Universal Robots PolyScope program: test1.urp

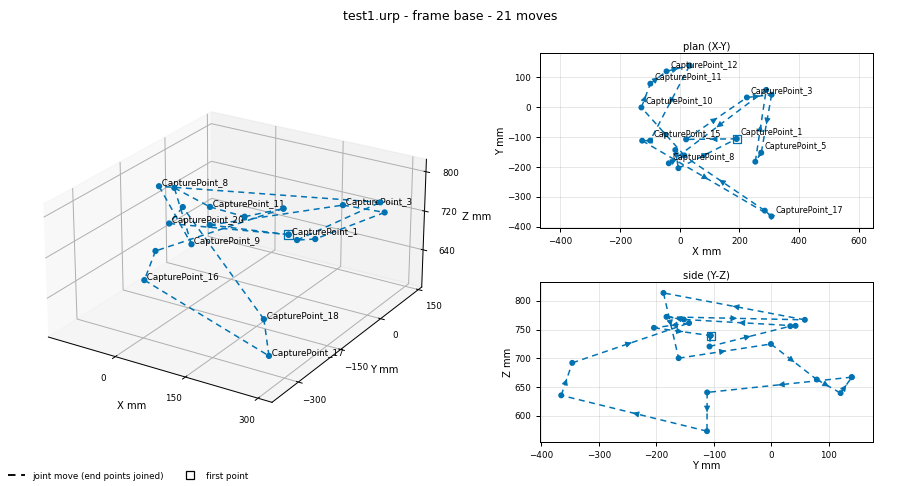
[picture p0: tool path of test1.urp in frame base, 21 of 21 moves have a stored position in this frame; points joined in program order, loops and branches not executed]
Program test1 (installation=default directory=/programs createdIn=3.8.0.61336 lastSavedIn=3.8.0.61336 robotSerialNumber=2018359174)
Calibrated DH parameters: a=[0.000103, -0.165236, -0.391809, -0.000008, 0.000072, 0]; d=[0.08937, 126.180413, -125.613724, -0.456703, 0.094787, 0.082637]; alpha=[1.569508, -0.003108, -0.027037, 1.57048, -1.570735, 0]; deltaTheta=[0, -1.172139, 1.133037, 0.038915, 0.000034, 0.000049]
Robot Program (runOnlyOnce=false)
  Script file /programs/X0.script
    | address="192.168.221.2"
    | port=3000
    | sname="mt"
    | socket_open(address,port,sname)
    | p=get_actual_tcp_pose()
    | socket_send_line("X0()",sname)
    | ret=socket_read_line(sname)
    | socket_close(sname)
    | if (ret != "OK"):
    |   popup(ret,title="X0",blocking=True)
    | end
  MoveJ speed 60 deg/s, acceleration 80 deg/s^2 (useActiveTCP=true)
    Waypoint CapturePoint_1: TCP in base x=190.534 y=-105.515 z=739.553 mm, rx=-2.169 ry=2.1248 rz=-0.0971 rad; joints [0.073, -70.662, -54.31, -138.22, 90.522, 0.198] deg
  Wait Sleep waitTime=1
  Script file /programs/X1.script
    | address="192.168.221.2"
    | port=3000
    | sname="mt"
    | socket_open(address,port,sname)
    | p=get_actual_tcp_pose()
    | rpy=rotvec2rpy([p[3],p[4],p[5]])
    | socket_send_string("X1(",sname)
    | socket_send_string(p[0]*1000.,sname)
    | socket_send_string(",",sname)
    | socket_send_string(p[1]*1000.,sname)
    | socket_send_string(",",sname)
    | socket_send_string(p[2]*1000.,sname)
    | socket_send_string(",",sname)
    | socket_send_string(r2d(rpy[0]),sname)
    | socket_send_string(",",sname)
    | socket_send_string(r2d(rpy[1]),sname)
    | socket_send_string(",",sname)
    | socket_send_string(r2d(rpy[2]),sname)
    | socket_send_line(")",sname)
    | ret=socket_read_line(sname)
    | socket_close(sname)
    | if (ret != "OK"):
    |   popup(ret,title="X1",blocking=True)
    | end
  MoveJ speed 60 deg/s, acceleration 80 deg/s^2 (useActiveTCP=true)
    Waypoint CapturePoint_2: TCP in base x=21.408 y=-107.346 z=720.582 mm, rx=-1.9877 ry=1.9105 rz=-0.2399 rad; joints [-30.105, -54.792, -66.384, -133.273, 107.073, -28.72] deg
  Wait Sleep waitTime=1
  Script file /programs/X1.script
    | (same text as the earlier copy of this file)
  MoveJ speed 60 deg/s, acceleration 80 deg/s^2 (useActiveTCP=true)
    Waypoint CapturePoint_3: TCP in base x=224.997 y=33.123 z=755.907 mm, rx=2.0802 ry=-2.0387 rz=0.3263 rad; joints [42.288, -80.135, -37.545, -164.25, 76.141, 44.096] deg
  Wait Sleep waitTime=1
  Script file /programs/X1.script
    | (same text as the earlier copy of this file)
  Wait Sleep waitTime=1
  MoveJ speed 60 deg/s, acceleration 80 deg/s^2 (useActiveTCP=true)
    Waypoint CapturePoint_4: TCP in base x=307.887 y=42.318 z=756.523 mm, rx=2.0137 ry=-1.9575 rz=0.3394 rad; joints [33.037, -92.913, -25.365, -167.152, 72.403, 35.309] deg
  Wait Sleep waitTime=1
  Script file /programs/X1.script
    | (same text as the earlier copy of this file)
  MoveJ speed 60 deg/s, acceleration 80 deg/s^2 (useActiveTCP=true)
    Waypoint CapturePoint_5: TCP in base x=273.105 y=-152.051 z=767.525 mm, rx=1.1431 ry=-2.8987 rz=-0.2387 rad; joints [-10.771, -92.914, -25.368, -157.055, 96.143, 37.312] deg
  Wait Sleep waitTime=1
  Script file /programs/X1.script
    | (same text as the earlier copy of this file)
  MoveJ speed 60 deg/s, acceleration 80 deg/s^2 (useActiveTCP=true)
    Waypoint CapturePoint_6: TCP in base x=253.251 y=-182.138 z=772.16 mm, rx=0.0328 ry=3.0997 rz=0.4007 rad; joints [-19.345, -92.915, -25.365, -155.309, 103.445, 72.846] deg
  Wait Sleep waitTime=1
  Script file /programs/X1.script
    | (same text as the earlier copy of this file)
  MoveJ speed 60 deg/s, acceleration 80 deg/s^2 (useActiveTCP=true)
    Waypoint CapturePoint_7: TCP in base x=289.745 y=58.466 z=766.928 mm, rx=2.7466 ry=0.3071 rz=0.0009 rad; joints [38.358, -91.191, -25.365, -165.797, 71.218, -60.862] deg
  Wait Sleep waitTime=1
  Script file /programs/X1.script
    | (same text as the earlier copy of this file)
  MoveJ speed 60 deg/s, acceleration 80 deg/s^2 (useActiveTCP=true)
    Waypoint CapturePoint_8: TCP in base x=-36.698 y=-187.426 z=813.704 mm, rx=-2.5132 ry=1.1035 rz=-0.5771 rad; joints [38.35, -58.013, -25.364, -158.36, 78.074, -5.557] deg
  Wait Sleep waitTime=1
  Script file /programs/X1.script
    | (same text as the earlier copy of this file)
  MoveJ speed 60 deg/s, acceleration 80 deg/s^2 (useActiveTCP=true)
    Waypoint CapturePoint_9: TCP in base x=15.55 y=-161.041 z=700.233 mm, rx=-2.5485 ry=1.1129 rz=-0.5577 rad; joints [43.689, -38.869, -67.087, -138.937, 75.373, -0.883] deg
  Wait Sleep waitTime=1
  Script file /programs/X1.script
    | (same text as the earlier copy of this file)
  MoveJ speed 60 deg/s, acceleration 80 deg/s^2 (useActiveTCP=true)
    Waypoint CapturePoint_10: TCP in base x=-128.422 y=-0.5 z=724.899 mm, rx=-1.2256 ry=2.2428 rz=-0.6001 rad; joints [-40.35, -38.871, -67.086, -127.735, 106.09, -0.879] deg
  Wait Sleep waitTime=1
  Script file /programs/X1.script
    | (same text as the earlier copy of this file)
  MoveJ speed 60 deg/s, acceleration 80 deg/s^2 (useActiveTCP=true)
    Waypoint CapturePoint_11: TCP in base x=-98.355 y=79.257 z=663.134 mm, rx=-0.6678 ry=2.3711 rz=-0.6414 rad; joints [-70.315, -30.072, -80.78, -124.448, 119.381, -0.99] deg
  Wait Sleep waitTime=1
  Script file /programs/X1.script
    | (same text as the earlier copy of this file)
  MoveJ speed 60 deg/s, acceleration 80 deg/s^2 (useActiveTCP=true)
    Waypoint CapturePoint_12: TCP in base x=-44.236 y=120.624 z=639.494 mm, rx=-0.028 ry=2.5208 rz=-0.5293 rad; joints [-97.846, -30.075, -80.778, -137.575, 123.899, -0.99] deg
  Wait Sleep waitTime=1
  Script file /programs/X1.script
    | (same text as the earlier copy of this file)
  MoveJ speed 60 deg/s, acceleration 80 deg/s^2 (useActiveTCP=true)
    Waypoint CapturePoint_13: TCP in base x=32.967 y=140.081 z=667.219 mm, rx=0.7689 ry=2.4403 rz=-0.2805 rad; joints [-127.955, -38.753, -66.496, -163.611, 124.333, -1.004] deg
  Wait Sleep waitTime=1
  Script file /programs/X1.script
    | (same text as the earlier copy of this file)
  MoveJ speed 60 deg/s, acceleration 80 deg/s^2 (useActiveTCP=true)
    Waypoint CapturePoint_14: TCP in base x=32.955 y=140.061 z=667.229 mm, rx=-1.0077 ry=2.5472 rz=-0.74 rad; joints [-127.955, -38.755, -66.496, -163.608, 124.335, -79.153] deg
  Wait Sleep waitTime=1
  Script file /programs/X1.script
    | (same text as the earlier copy of this file)
  MoveJ speed 60 deg/s, acceleration 80 deg/s^2 (useActiveTCP=true)
    Waypoint CapturePoint_15: TCP in base x=-98.976 y=-111.429 z=640.718 mm, rx=-1.9221 ry=1.7558 rz=-0.7168 rad; joints [0.392, -27.054, -85.502, -117.851, 86.877, -4.56] deg
  Wait Sleep waitTime=1
  Script file /programs/X1.script
    | (same text as the earlier copy of this file)
  MoveJ speed 60 deg/s, acceleration 80 deg/s^2 (useActiveTCP=true)
    Waypoint CapturePoint_16: TCP in base x=-125.724 y=-111.715 z=573.266 mm, rx=-1.7134 ry=1.786 rz=-0.7532 rad; joints [0.402, -15.524, -97.784, -110.625, 86.851, 2.752] deg
  Wait Sleep waitTime=1
  Script file /programs/X1.script
    | (same text as the earlier copy of this file)
  MoveJ speed 60 deg/s, acceleration 80 deg/s^2 (useActiveTCP=true)
    Waypoint CapturePoint_17: TCP in base x=307.338 y=-365.217 z=635.603 mm, rx=-1.8392 ry=1.9097 rz=0.7596 rad; joints [-40.903, -107.911, -31.186, -161.588, 113.228, -43.898] deg
  Wait Sleep waitTime=1
  Script file /programs/X1.script
    | (same text as the earlier copy of this file)
  MoveJ speed 60 deg/s, acceleration 80 deg/s^2 (useActiveTCP=true)
    Waypoint CapturePoint_18: TCP in base x=285.042 y=-346.037 z=692.112 mm, rx=-0.2019 ry=-2.9931 rz=-0.8493 rad; joints [-40.903, -107.916, -21.263, -161.588, 113.234, 53.855] deg
  Wait Sleep waitTime=1
  Script file /programs/X1.script
    | (same text as the earlier copy of this file)
  MoveJ speed 60 deg/s, acceleration 80 deg/s^2 (useActiveTCP=true)
    Waypoint CapturePoint_19: TCP in base x=-14.788 y=-142.877 z=761.304 mm, rx=0.9846 ry=2.4689 rz=0.6334 rad; joints [-71.114, -70.355, -47.356, -156.575, 124.411, 62.513] deg
  Wait Sleep waitTime=1
  Script file /programs/X1.script
    | (same text as the earlier copy of this file)
  MoveJ speed 60 deg/s, acceleration 80 deg/s^2 (useActiveTCP=true)
    Waypoint CapturePoint_20: TCP in base x=-4.371 y=-203.918 z=753.086 mm, rx=-1.8631 ry=1.8783 rz=-0.0962 rad; joints [-71.114, -77.335, -43.394, -157.914, 116.465, -71.239] deg
  Wait Sleep waitTime=1
  Script file /programs/X1.script
    | (same text as the earlier copy of this file)
  MoveJ speed 60 deg/s, acceleration 80 deg/s^2 (useActiveTCP=true)
    Waypoint CapturePoint_1: TCP in base x=190.534 y=-105.515 z=739.553 mm, rx=-2.169 ry=2.1248 rz=-0.0971 rad; joints [0.073, -70.662, -54.31, -138.22, 90.522, 0.198] deg
  Script file /programs/X2-rcalib.script
    | address="192.168.221.2"
    | port=3000
    | sname="mt"
    | socket_open(address,port,sname)
    | p=get_actual_tcp_pose()
    | socket_send_line("X2()",sname)
    | ret=socket_read_line(sname)
    | socket_close(sname)
  Halt
